{attribute 'qualified_only'}
VAR_GLOBAL
	mb_Input_Coils    		:    ARRAY [0..255] OF BOOL;
	mb_Output_Coils 		:    ARRAY [0..255] OF BOOL;
	mb_Input_Registers 		:    ARRAY [0..255] OF WORD;
	mb_Output_Registers 	:    ARRAY [0..255] OF WORD;
END_VAR

(* stored: Version 1.1.0.1, ProductVersion 3.1.4024.12
   GVL GVL: Id {1491c449-ef4f-4bea-8942-80bc0e7a5008} *)
